Fanuc KAREL source: kb00111.KL

-- PROVISIONAL review KL for V940-1; original PC SHA256 cf512adf2a9857eca1666f7e598325e32b3bdcdd6765d20d5e397984ff477a4a
-- Incomplete behavior may be omitted. Consult companion uncertainty JSON. Do not deploy.
PROGRAM KB00111
%NOLOCKGROUP
BEGIN
  -- V9_ZERO_TABLE_METADATA_HINT layout=0002_ascii; no indexed target words; source/name/runtime held
  -- UNRESOLVED_PC offsets 5-21; opcodes 27,22,31,23
  -- UNRESOLVED_PC offsets 26-30; opcodes 7F
END KB00111
